(* Logix 5000 project; controller Drives_Line1 1756-L72 rev 20.13; software revision 20.04; part 5 of 21 *)
(* tags used below, declared in another part *)
   Diamtest : BOOL;
   Diamtest_mm : REAL;
   TimeForBr : TIMER;
   TimeOffFan : TIMER;
   TonRefOn : TIMER;
   Unwinder_1_DiamCalcOn : BOOL;
   Unwinder_1_JEC : REAL;
   Unwinder_1_JLossCrvSpd : REAL[21];
   Unwinder_1_JMaterial : REAL;
   Unwinder_1_LossCrvTrq_Pct : REAL[21];
   Unwinder_1_MatMass : REAL;
   Unwinder_1_MatVolume : REAL;
   Unwinder_1_MaxMass : REAL;
   Unwinder_1_MaxVolume : REAL;
   Unwinder_1_PctPerN : REAL;
   Unwinder_1_RatedTrq : REAL;
   Unwinder_1_RPMPerMPS : REAL;
   Unwinder_1_Running : BOOL;
   Unwinder_1_SpdMps_Flt : REAL;
   Unwinder_1_SpdRpm_Flt : REAL;
   zUnwinder_1_JGainQ1Q2 : REAL;
   zUnwinder_1_JGainQ3Q4 : REAL;
   zUnwinder_1_RateMax : REAL;
   zUnwinder_1_SpdReg_BWMax : REAL;
   zUnwinder_1_SpdReg_BWmin : REAL;
   zUnwinder_1_Stall_Spd : REAL;
   zUnwinder_1_TenRefRate : REAL;
   zUnwinder_1_TenSpStall : REAL;
   zUnwinder_1_TrqTrimLimMax_Pct : REAL;
   zUnwinder_1_TrqTrimLimMin_Pct : REAL;
   Bridle_01 : UDT_Bridle_3M;
   EntryConfig : UDT_Config_Zone;
   EntryCtrl : UDT_Control_Zone;
   LineSetpoints : UDT_Setpoints_Line;
   Unwinder_1 : UDT_Unwinder;
   Winder : UDT_Winder;
   zPi : REAL;
(* P10_Unwinder_1, continued *)

ROUTINE R05_Control   (* ladder *)
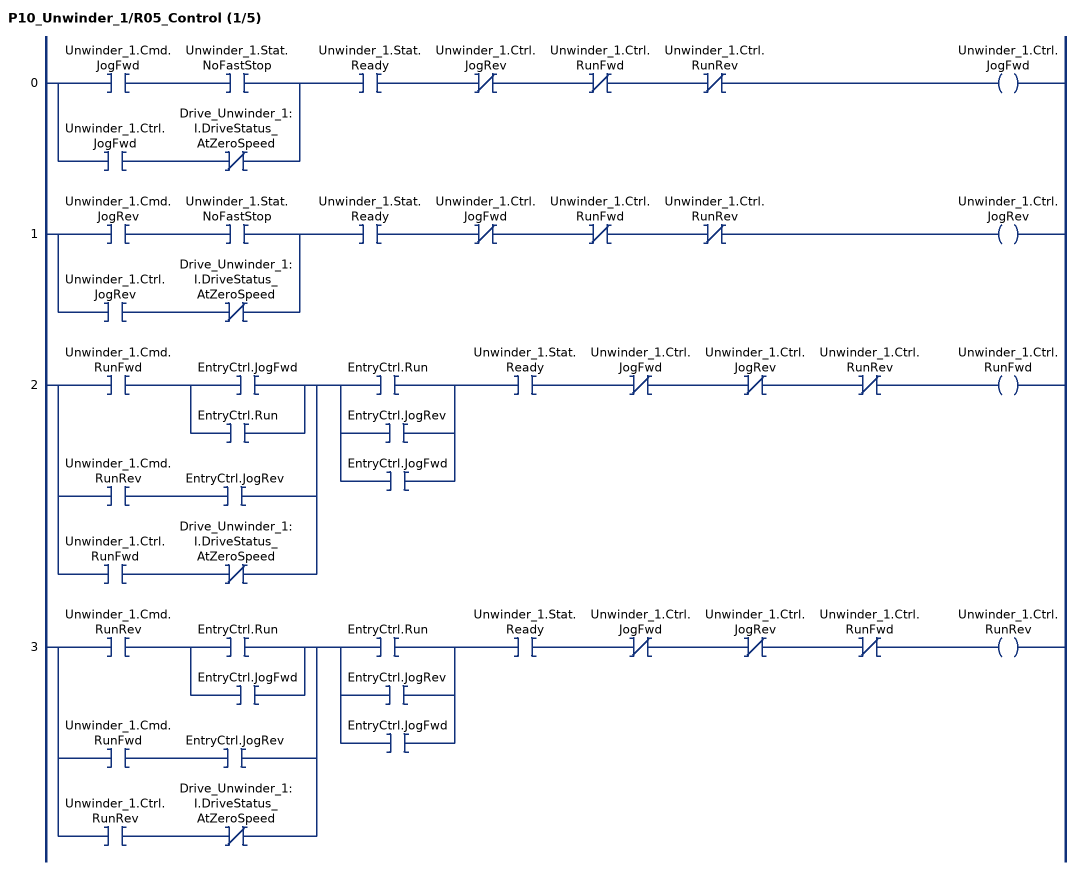
   0: [XIC(Unwinder_1.Cmd.JogFwd) XIC(Unwinder_1.Stat.NoFastStop) ,XIC(Unwinder_1.Ctrl.JogFwd) XIO(Drive_Unwinder_1:I.DriveStatus_AtZeroSpeed) ]XIC(Unwinder_1.Stat.Ready)XIO(Unwinder_1.Ctrl.JogRev)XIO(Unwinder_1.Ctrl.RunFwd)XIO(Unwinder_1.Ctrl.RunRev)OTE(Unwinder_1.Ctrl.JogFwd);
   1: [XIC(Unwinder_1.Cmd.JogRev) XIC(Unwinder_1.Stat.NoFastStop) ,XIC(Unwinder_1.Ctrl.JogRev) XIO(Drive_Unwinder_1:I.DriveStatus_AtZeroSpeed) ]XIC(Unwinder_1.Stat.Ready)XIO(Unwinder_1.Ctrl.JogFwd)XIO(Unwinder_1.Ctrl.RunFwd)XIO(Unwinder_1.Ctrl.RunRev)OTE(Unwinder_1.Ctrl.JogRev);
   2: [XIC(Unwinder_1.Cmd.RunFwd) [XIC(EntryCtrl.JogFwd) ,XIC(EntryCtrl.Run) ] ,XIC(Unwinder_1.Cmd.RunRev) XIC(EntryCtrl.JogRev) ,XIC(Unwinder_1.Ctrl.RunFwd) XIO(Drive_Unwinder_1:I.DriveStatus_AtZeroSpeed) ][XIC(EntryCtrl.Run) ,XIC(EntryCtrl.JogRev) ,XIC(EntryCtrl.JogFwd) ]XIC(Unwinder_1.Stat.Ready)XIO(Unwinder_1.Ctrl.JogFwd)XIO(Unwinder_1.Ctrl.JogRev)XIO(Unwinder_1.Ctrl.RunRev)OTE(Unwinder_1.Ctrl.RunFwd);
   3: [XIC(Unwinder_1.Cmd.RunRev) [XIC(EntryCtrl.Run) ,XIC(EntryCtrl.JogFwd) ] ,XIC(Unwinder_1.Cmd.RunFwd) XIC(EntryCtrl.JogRev) ,XIC(Unwinder_1.Ctrl.RunRev) XIO(Drive_Unwinder_1:I.DriveStatus_AtZeroSpeed) ][XIC(EntryCtrl.Run) ,XIC(EntryCtrl.JogRev) ,XIC(EntryCtrl.JogFwd) ]XIC(Unwinder_1.Stat.Ready)XIO(Unwinder_1.Ctrl.JogFwd)XIO(Unwinder_1.Ctrl.JogRev)XIO(Unwinder_1.Ctrl.RunFwd)OTE(Unwinder_1.Ctrl.RunRev);
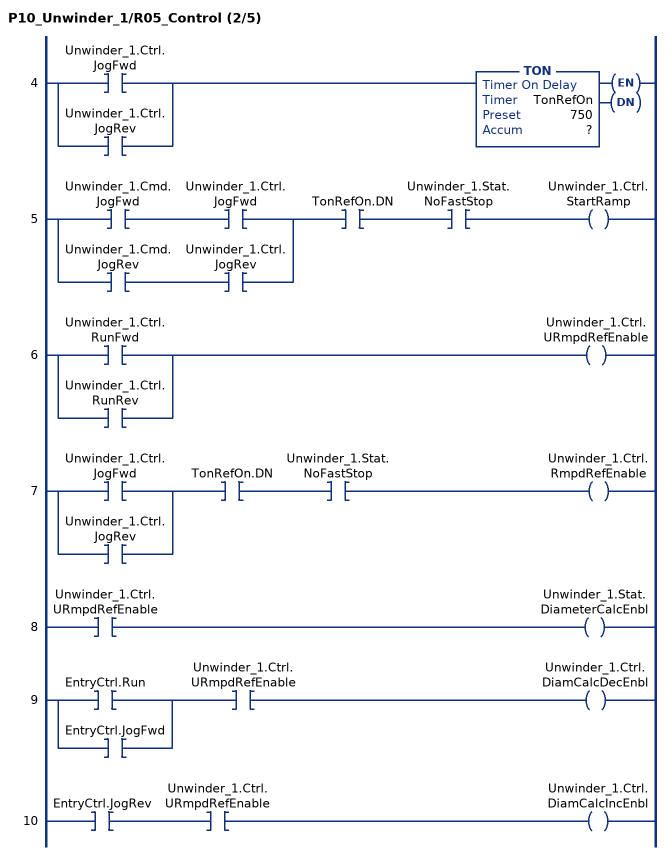
   4: [XIC(Unwinder_1.Ctrl.JogFwd) ,XIC(Unwinder_1.Ctrl.JogRev) ]TON(TonRefOn,?,?);
   5: [XIC(Unwinder_1.Cmd.JogFwd) XIC(Unwinder_1.Ctrl.JogFwd) ,XIC(Unwinder_1.Cmd.JogRev) XIC(Unwinder_1.Ctrl.JogRev) ]XIC(TonRefOn.DN)XIC(Unwinder_1.Stat.NoFastStop)OTE(Unwinder_1.Ctrl.StartRamp);
   6: [XIC(Unwinder_1.Ctrl.RunFwd) ,XIC(Unwinder_1.Ctrl.RunRev) ]OTE(Unwinder_1.Ctrl.URmpdRefEnable);
   7: [XIC(Unwinder_1.Ctrl.JogFwd) ,XIC(Unwinder_1.Ctrl.JogRev) ]XIC(TonRefOn.DN)XIC(Unwinder_1.Stat.NoFastStop)OTE(Unwinder_1.Ctrl.RmpdRefEnable);
   8: XIC(Unwinder_1.Ctrl.URmpdRefEnable)OTE(Unwinder_1.Stat.DiameterCalcEnbl);
   9: [XIC(EntryCtrl.Run) ,XIC(EntryCtrl.JogFwd) ]XIC(Unwinder_1.Ctrl.URmpdRefEnable)OTE(Unwinder_1.Ctrl.DiamCalcDecEnbl);
   10: XIC(EntryCtrl.JogRev)XIC(Unwinder_1.Ctrl.URmpdRefEnable)OTE(Unwinder_1.Ctrl.DiamCalcIncEnbl);
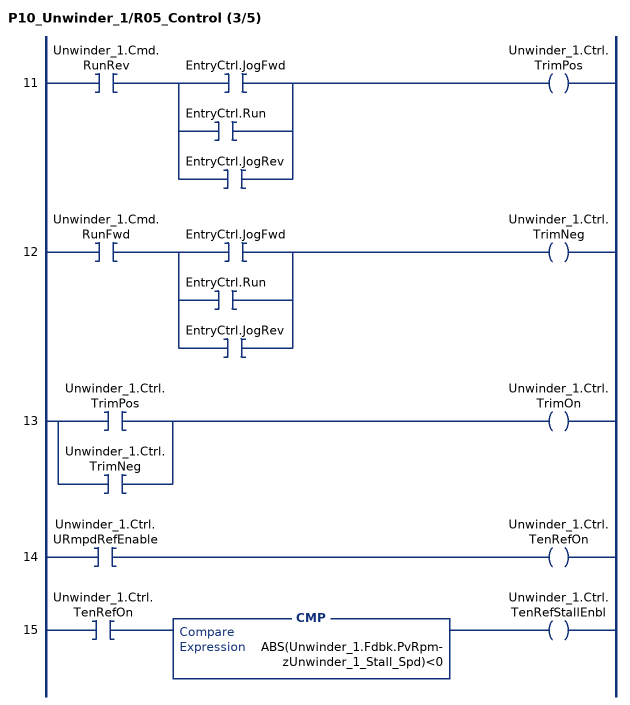
   11: XIC(Unwinder_1.Cmd.RunRev)[XIC(EntryCtrl.JogFwd) ,XIC(EntryCtrl.Run) ,XIC(EntryCtrl.JogRev) ]OTE(Unwinder_1.Ctrl.TrimPos);
   12: XIC(Unwinder_1.Cmd.RunFwd)[XIC(EntryCtrl.JogFwd) ,XIC(EntryCtrl.Run) ,XIC(EntryCtrl.JogRev) ]OTE(Unwinder_1.Ctrl.TrimNeg);
   13: [XIC(Unwinder_1.Ctrl.TrimPos) ,XIC(Unwinder_1.Ctrl.TrimNeg) ]OTE(Unwinder_1.Ctrl.TrimOn);
   14: XIC(Unwinder_1.Ctrl.URmpdRefEnable)OTE(Unwinder_1.Ctrl.TenRefOn);
   15: XIC(Unwinder_1.Ctrl.TenRefOn)CMP(ABS(Unwinder_1.Fdbk.PvRpm-zUnwinder_1_Stall_Spd)<0)OTE(Unwinder_1.Ctrl.TenRefStallEnbl);
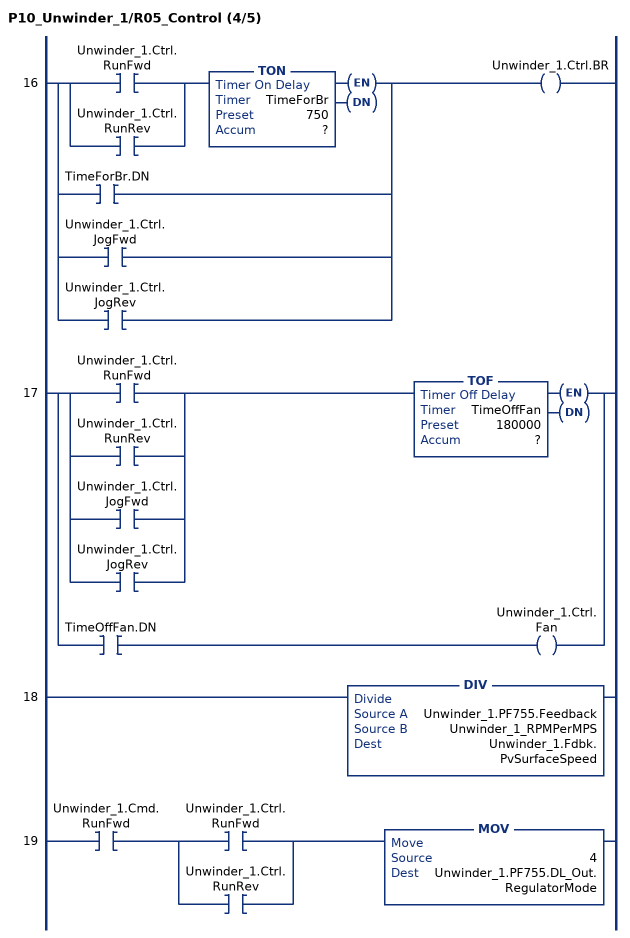
   16: [[XIC(Unwinder_1.Ctrl.RunFwd) ,XIC(Unwinder_1.Ctrl.RunRev) ] TON(TimeForBr,?,?) ,XIC(TimeForBr.DN) ,XIC(Unwinder_1.Ctrl.JogFwd) ,XIC(Unwinder_1.Ctrl.JogRev) ]OTE(Unwinder_1.Ctrl.BR);
   17: [[XIC(Unwinder_1.Ctrl.RunFwd) ,XIC(Unwinder_1.Ctrl.RunRev) ,XIC(Unwinder_1.Ctrl.JogFwd) ,XIC(Unwinder_1.Ctrl.JogRev) ] TOF(TimeOffFan,?,?) ,XIC(TimeOffFan.DN) OTE(Unwinder_1.Ctrl.Fan) ];
   18: DIV(Unwinder_1.PF755.Feedback,Unwinder_1_RPMPerMPS,Unwinder_1.Fdbk.PvSurfaceSpeed);
   19: XIC(Unwinder_1.Cmd.RunFwd)[XIC(Unwinder_1.Ctrl.RunFwd) ,XIC(Unwinder_1.Ctrl.RunRev) ]MOV(4,Unwinder_1.PF755.DL_Out.RegulatorMode);
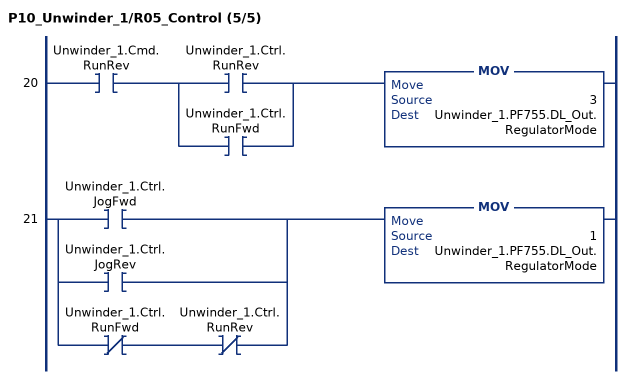
   20: XIC(Unwinder_1.Cmd.RunRev)[XIC(Unwinder_1.Ctrl.RunRev) ,XIC(Unwinder_1.Ctrl.RunFwd) ]MOV(3,Unwinder_1.PF755.DL_Out.RegulatorMode);
   21: [XIC(Unwinder_1.Ctrl.JogFwd) ,XIC(Unwinder_1.Ctrl.JogRev) ,XIO(Unwinder_1.Ctrl.RunFwd) XIO(Unwinder_1.Ctrl.RunRev) ]MOV(1,Unwinder_1.PF755.DL_Out.RegulatorMode);
END_ROUTINE

ROUTINE R07_TenFb   (* function block diagram *)
   SHEET 1   // Torque Feedback
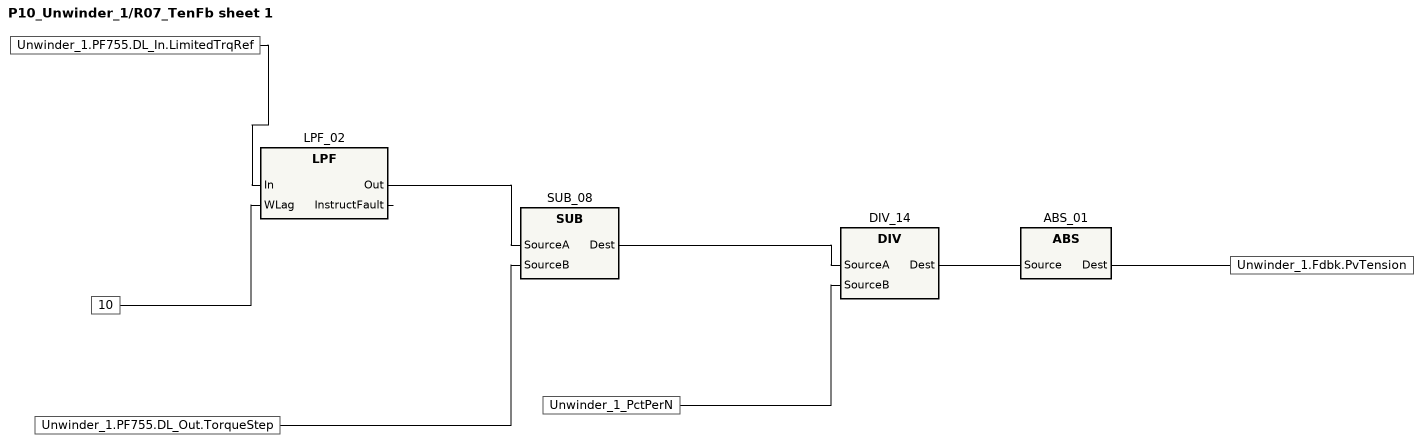
   LPF_02 : LPF(In := Unwinder_1.PF755.DL_In.LimitedTrqRef, WLag := 10);   // unwired pins: InstructFault
   SUB_08 : SUB(SourceA := LPF_02.Out, SourceB := Unwinder_1.PF755.DL_Out.TorqueStep);
   DIV_14 : DIV(SourceA := SUB_08.Dest, SourceB := Unwinder_1_PctPerN);
   ABS_01 : ABS(Source := DIV_14.Dest);
   Unwinder_1.Fdbk.PvTension := ABS_01.Dest;
   SHEET 2   // Speed Feedback
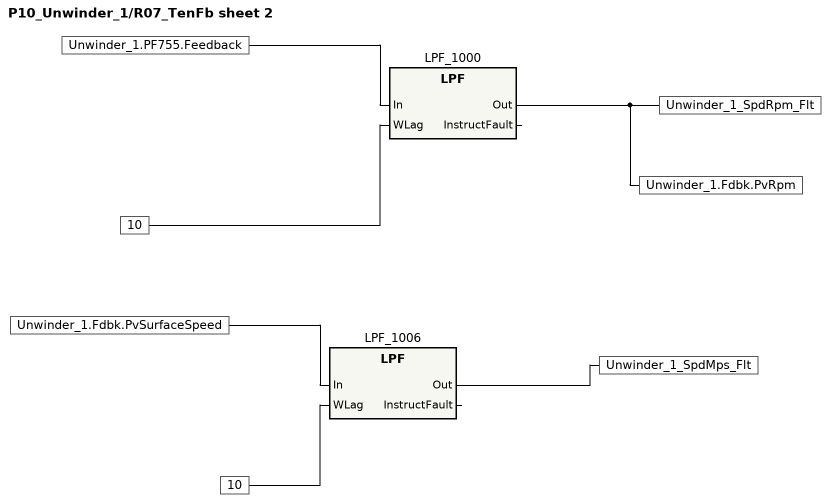
   LPF_1006 : LPF(In := Unwinder_1.Fdbk.PvSurfaceSpeed, WLag := 10);   // unwired pins: InstructFault
   LPF_1000 : LPF(In := Unwinder_1.PF755.Feedback, WLag := 10);   // unwired pins: InstructFault
   Unwinder_1_SpdMps_Flt := LPF_1006.Out;
   Unwinder_1.Fdbk.PvRpm := LPF_1000.Out;
   Unwinder_1_SpdRpm_Flt := LPF_1000.Out;
END_ROUTINE

ROUTINE R09_DiamCalc   (* function block diagram *)
   SHEET 1   // Distance/Angle Integration
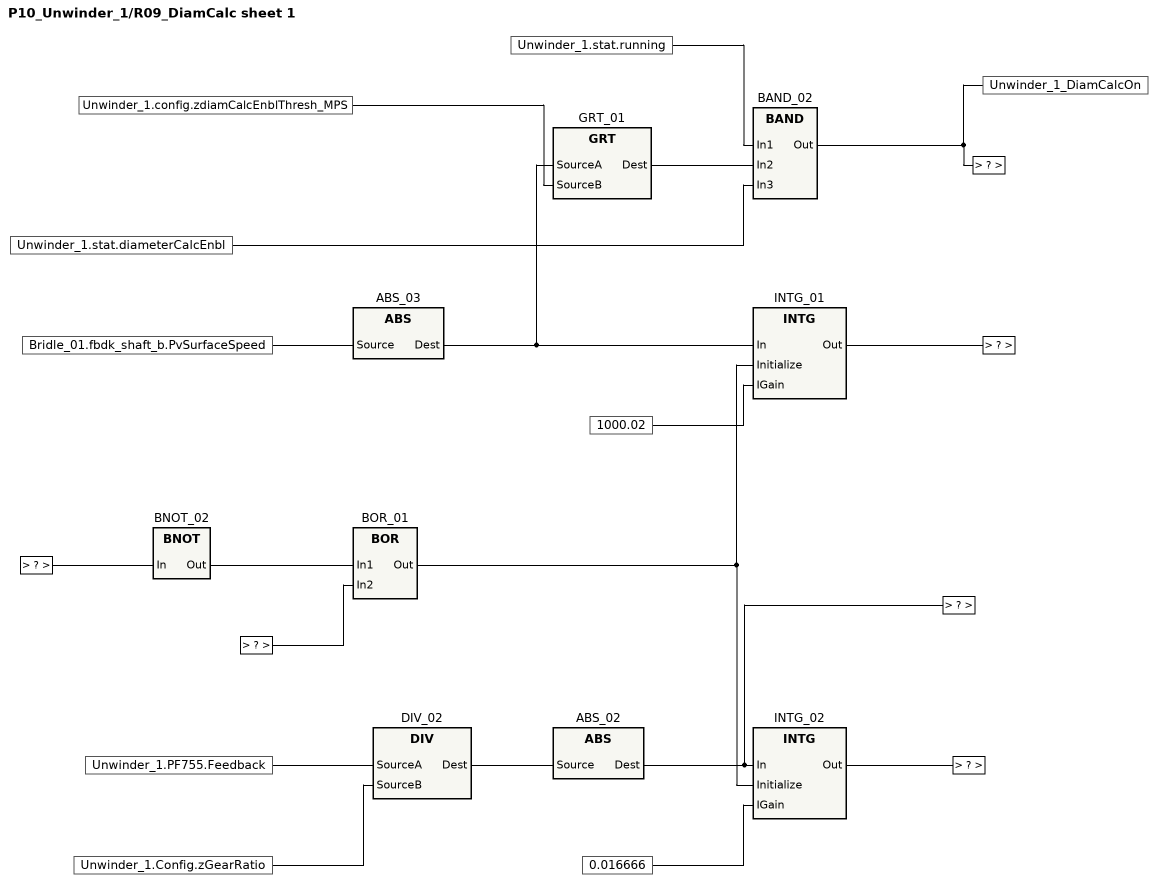
   ABS_03 : ABS(Source := Bridle_01.fbdk_shaft_b.PvSurfaceSpeed);
   DIV_02 : DIV(SourceA := Unwinder_1.PF755.Feedback, SourceB := Unwinder_1.Config.zGearRatio);
   GRT_01 : GRT(SourceA := ABS_03.Dest, SourceB := Unwinder_1.config.zdiamCalcEnblThresh_MPS);
   ABS_02 : ABS(Source := DIV_02.Dest);
   BAND_02 : BAND(In1 := Unwinder_1.stat.running, In2 := GRT_01.Dest, In3 := Unwinder_1.stat.diameterCalcEnbl);
   WIRE(?) := ABS_02.Dest;
   BNOT_02 : BNOT(In := WIRE(?));
   BOR_01 : BOR(In1 := BNOT_02.Out, In2 := WIRE(?) {feedback});
   INTG_01 : INTG(In := ABS_03.Dest, Initialize := BOR_01.Out, IGain := 1000.02);
   INTG_02 : INTG(In := ABS_02.Dest, Initialize := BOR_01.Out, IGain := 0.016666);
   WIRE(?) := INTG_02.Out;
   WIRE(?) := BAND_02.Out;
   Unwinder_1_DiamCalcOn := BAND_02.Out;
   WIRE(?) := INTG_01.Out;
   SHEET 2   // Diameter Calculate
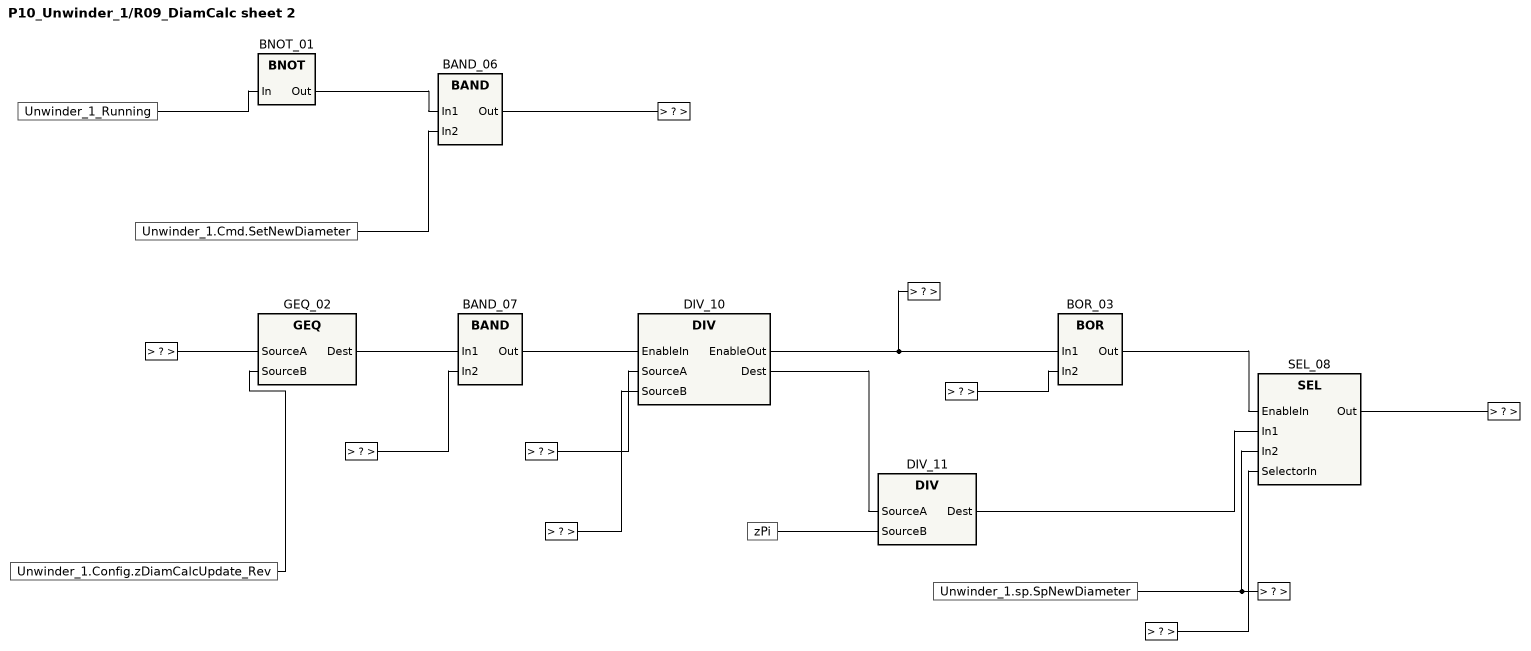
   BNOT_01 : BNOT(In := Unwinder_1_Running);
   BAND_06 : BAND(In1 := BNOT_01.Out, In2 := Unwinder_1.Cmd.SetNewDiameter);
   WIRE(?) := BAND_06.Out;
   WIRE(?) := Unwinder_1.sp.SpNewDiameter;
   GEQ_02 : GEQ(SourceA := WIRE(?), SourceB := Unwinder_1.Config.zDiamCalcUpdate_Rev);
   BAND_07 : BAND(In1 := GEQ_02.Dest, In2 := WIRE(?));
   DIV_10 : DIV(EnableIn := BAND_07.Out, SourceA := WIRE(?), SourceB := WIRE(?));
   DIV_11 : DIV(SourceA := DIV_10.Dest, SourceB := zPi);
   WIRE(?) := DIV_10.EnableOut;
   BOR_03 : BOR(In1 := DIV_10.EnableOut, In2 := WIRE(?));
   SEL_08 : SEL(EnableIn := BOR_03.Out, In1 := DIV_11.Dest, In2 := Unwinder_1.sp.SpNewDiameter, SelectorIn := WIRE(?));
   WIRE(?) := SEL_08.Out;
   SHEET 3   // Rate/Magnitude Limit
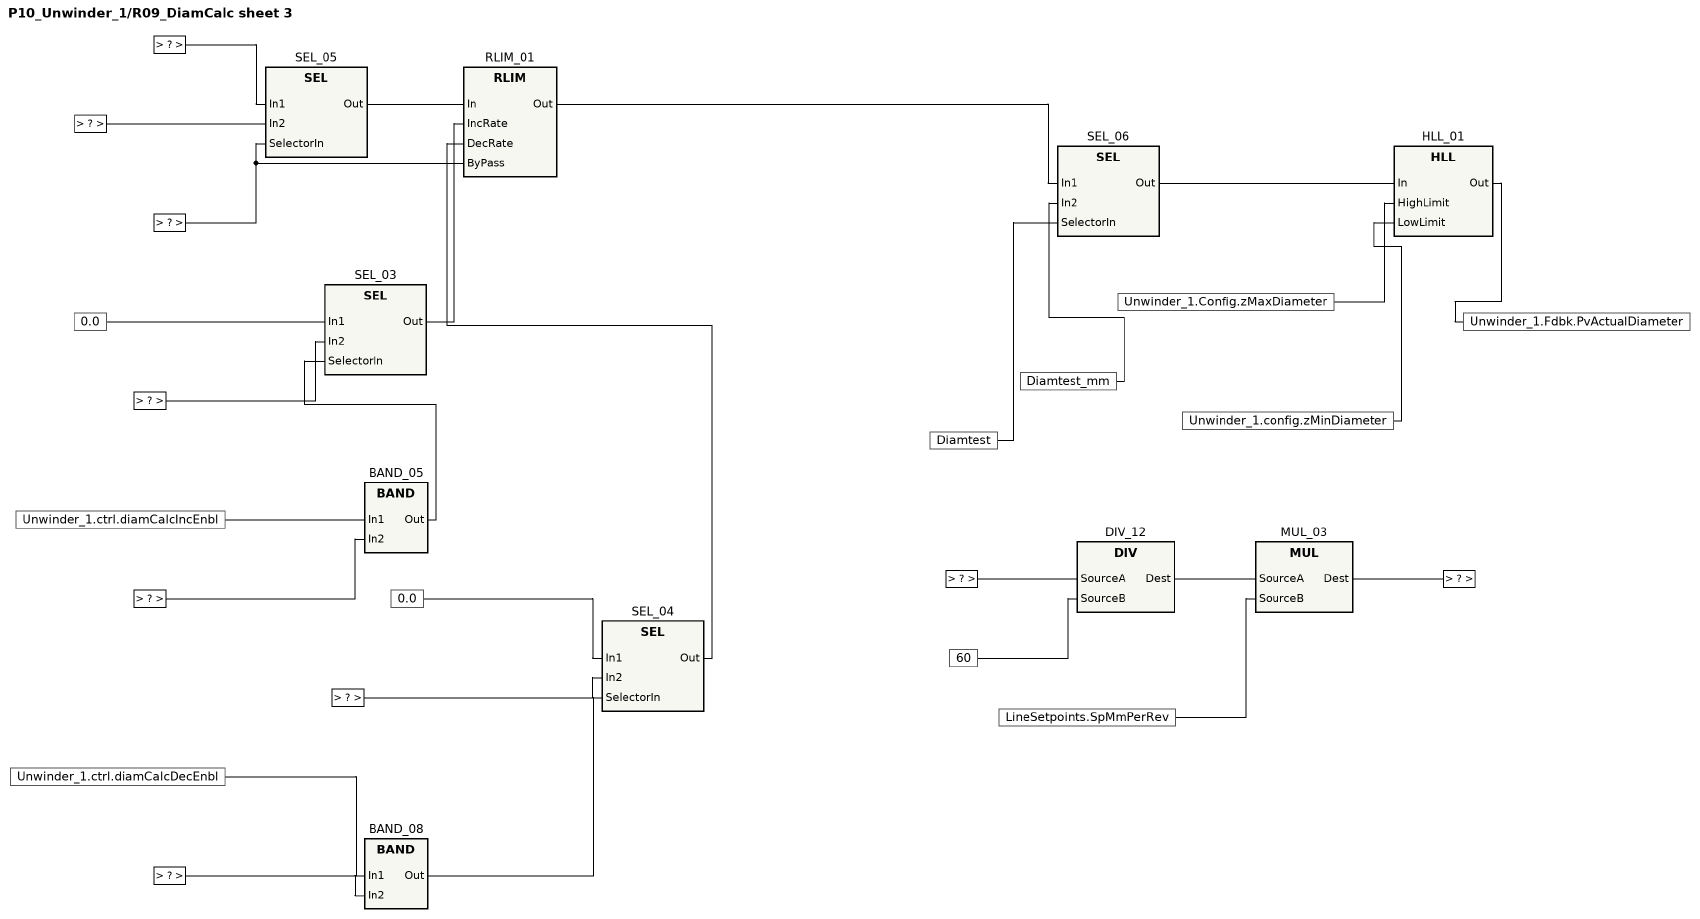
   BAND_05 : BAND(In1 := Unwinder_1.ctrl.diamCalcIncEnbl, In2 := WIRE(?));
   SEL_03 : SEL(In1 := 0.0, In2 := WIRE(?), SelectorIn := BAND_05.Out);
   SEL_05 : SEL(In1 := WIRE(?), In2 := WIRE(?), SelectorIn := WIRE(?));
   BAND_08 : BAND(In1 := Unwinder_1.ctrl.diamCalcDecEnbl, In2 := WIRE(?));
   SEL_04 : SEL(In1 := 0.0, In2 := WIRE(?), SelectorIn := BAND_08.Out);
   RLIM_01 : RLIM(In := SEL_05.Out, IncRate := SEL_03.Out, DecRate := SEL_04.Out, ByPass := WIRE(?));
   SEL_06 : SEL(In1 := RLIM_01.Out, In2 := Diamtest_mm, SelectorIn := Diamtest);
   HLL_01 : HLL(In := SEL_06.Out, HighLimit := Unwinder_1.Config.zMaxDiameter, LowLimit := Unwinder_1.config.zMinDiameter);
   Unwinder_1.Fdbk.PvActualDiameter := HLL_01.Out;
   DIV_12 : DIV(SourceA := WIRE(?), SourceB := 60);
   MUL_03 : MUL(SourceA := DIV_12.Dest, SourceB := LineSetpoints.SpMmPerRev);
   WIRE(?) := MUL_03.Dest;
END_ROUTINE

ROUTINE R10_Calculate   (* structured text *)
   // Calculate
   // Speed Conversion
   //
   // * * * * * * * * * * * * * * * * * * * * * * * * * * *
   //
   // Calculates conversion factor from surface speed [MPS] to rotational speeds [RPM].
   //
   //             Gear Ratio * 1000 [mm/M]
   // RPM/MPS =  -------------------------- * 60
   //             Roll Diameter [mm] * PI
   //
   Unwinder_1_RPMPerMPS := (Unwinder_1.Config.zGearRatio * 1000.0) / (Unwinder_1.Fdbk.PvActualDiameter * zPi) * 60;
   //
   // * * * * * * * * * * * * * * * * * * * * * * * * * * *
   //
   // Calculate
   // (Rated Motor Torque)
   //
   // * * * * * * * * * * * * * * * * * * * * * * * * * * *
   //
   //                       MtrPwrRated [KW] * 9549
   // MtrTrqRated_Nm = ----------------------------
   //                           MtrSpdBase [RPM]
   //
   Unwinder_1_RatedTrq := Unwinder_1.Config.zMotorPwr * 9549 / Unwinder_1.Config.zMtrBaseSpd;
   //
   
   
   //
   // Calculate
   // (Center Winder Inertia)
   //
   // * * * * * * * * * * * * * * * * * * * * * * * * * * *
   //
   // MaterialVolume_m3 = (Pi * (Diam_mm/2000)**2 - Pi * (DiamMinEC_mm/2000)**2) * Width_mm/1000
   //
   Unwinder_1_MatVolume := (zPi * (Unwinder_1.Fdbk.PvActualDiameter/2000)**2)
   - (zPi * (Unwinder_1.Config.zMinDiameter/2000)**2)* (LineSetpoints.WebWidth  / 1000);
   Unwinder_1_MaxVolume:= (zPi * (Unwinder_1.Config.zMaxDiameter/2000)**2)* LineSetpoints.WebWidth / 1000;
   // MaterialMass_Kg = MaterialVolume_m3 * Density_Kgm3
   //
   Unwinder_1_MatMass := Unwinder_1_MatVolume * LineSetpoints.MaterialDensity ;
   Unwinder_1_MaxMass:= Unwinder_1_MaxVolume * LineSetpoints.MaterialDensity ;
   //
   // JMaterial_Kgm2 = MaterialWeight_Kg / 2 * ((Diam_mm/2000)**2 + (DiamMinEC_mm/2000)**2) / GearRatio**2
   //
   Unwinder_1_JMaterial := Unwinder_1_MatMass / 2 *
   ((Unwinder_1.Fdbk.PvActualDiameter/2000)**2 + (Unwinder_1.Config.zMinDiameter/2000)**2)
    / Unwinder_1.Config.zGearRatio**2 ;
   //
   // Calculate total reflected inertia [kilogram-meters**2]
   //
   Unwinder_1.Fdbk.PvTotalInertia := Unwinder_1_JEC + Unwinder_1_JMaterial ;
   //
   // * * * * * * * * * * * * * * * * * * * * * * * * * * *
   //
   // Calculate
   // (Normalized Inertia)
   //
   // * * * * * * * * * * * * * * * * * * * * * * * * * * *
   //
   //         J [Kgm**2] * MtrSpdBase [RPM]
   // J_Sec = -------------------------------
   //           9.549 * MtrTrqRated [Nm]
   //
   Unwinder_1.Fdbk.PvNormInertia := (Unwinder_1.Fdbk.PvTotalInertia * Unwinder_1.Config.zMtrBaseSpd)
   / (9.549 * Unwinder_1_RatedTrq);
   
   (*                         Diam [mm]           100                  1      *)
   (* Conversion_PctPerN =  ----------- * -------------------- * ----------- *)
   (*                         1000 * 2       MtrTrqRated [Nm]      GearRatio  *)
   
   Unwinder_1_PctPerN := Unwinder_1.Fdbk.PvActualDiameter / Unwinder_1.Config.zGearRatio
    / Unwinder_1_RatedTrq / 20.0 ;
END_ROUTINE

ROUTINE R11_TenRef   (* function block diagram *)
   SHEET 1   // Tension Reference
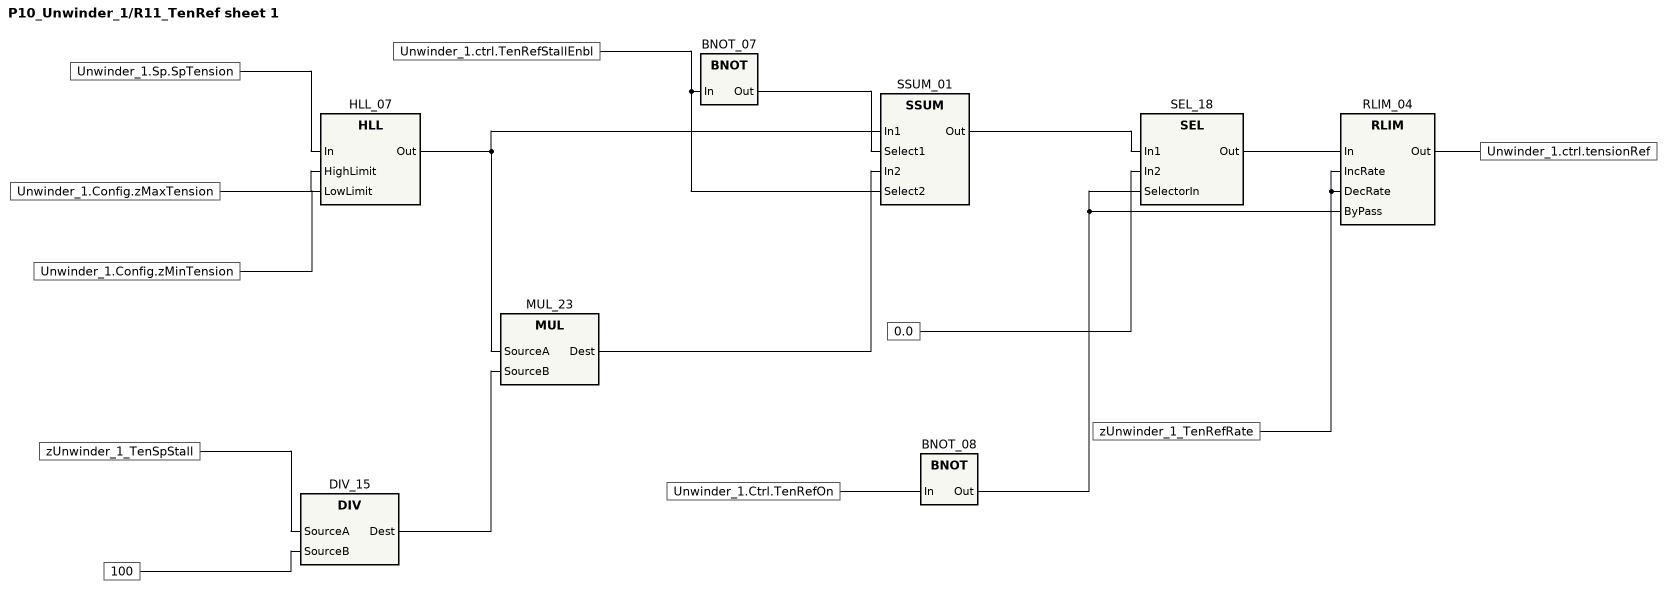
   DIV_15 : DIV(SourceA := zUnwinder_1_TenSpStall, SourceB := 100);
   HLL_07 : HLL(In := Unwinder_1.Sp.SpTension, HighLimit := Unwinder_1.Config.zMaxTension, LowLimit := Unwinder_1.Config.zMinTension);
   MUL_23 : MUL(SourceA := HLL_07.Out, SourceB := DIV_15.Dest);
   BNOT_07 : BNOT(In := Unwinder_1.ctrl.TenRefStallEnbl);
   SSUM_01 : SSUM(In1 := HLL_07.Out, Select1 := BNOT_07.Out, In2 := MUL_23.Dest, Select2 := Unwinder_1.ctrl.TenRefStallEnbl);
   BNOT_08 : BNOT(In := Unwinder_1.Ctrl.TenRefOn);
   SEL_18 : SEL(In1 := SSUM_01.Out, In2 := 0.0, SelectorIn := BNOT_08.Out);
   RLIM_04 : RLIM(In := SEL_18.Out, IncRate := zUnwinder_1_TenRefRate, DecRate := zUnwinder_1_TenRefRate, ByPass := BNOT_08.Out);
   Unwinder_1.ctrl.tensionRef := RLIM_04.Out;
END_ROUTINE

ROUTINE R12_DriveRef   (* function block diagram *)
   SHEET 1   // Jog reference
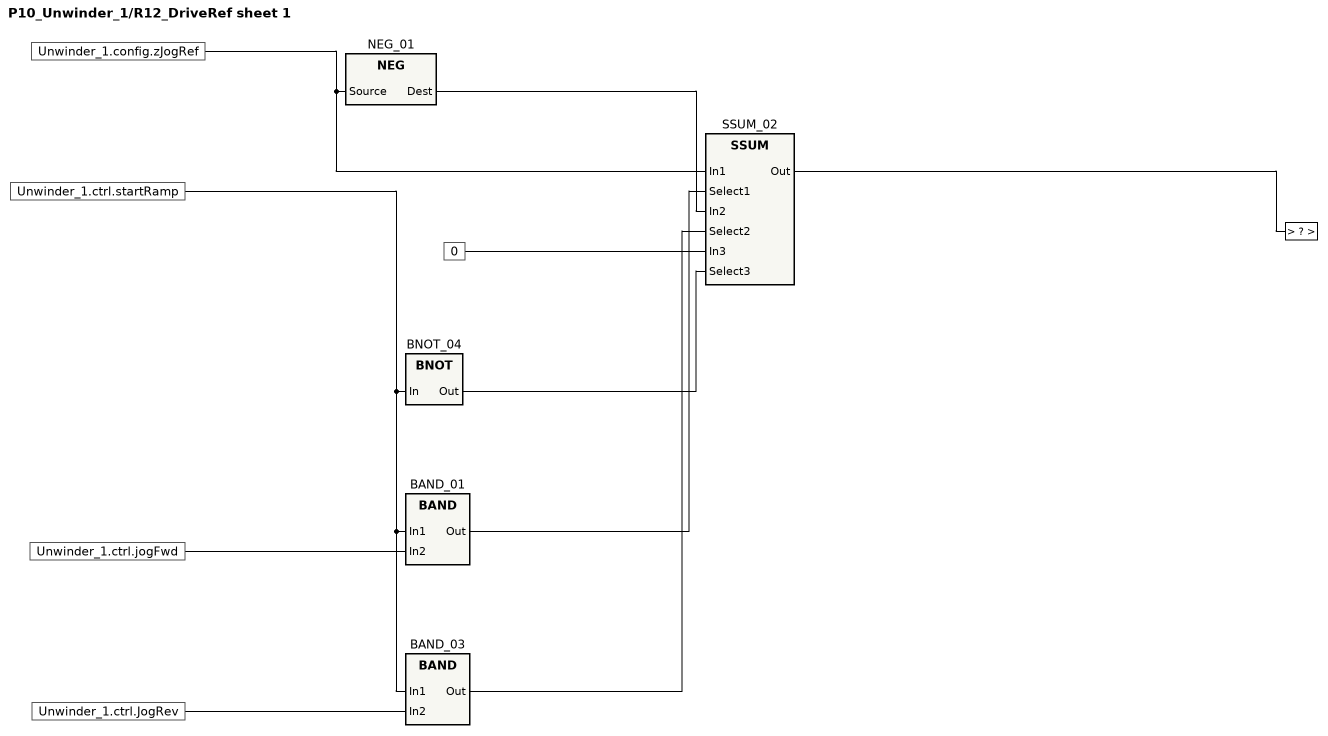
   NEG_01 : NEG(Source := Unwinder_1.config.zJogRef);
   BNOT_04 : BNOT(In := Unwinder_1.ctrl.startRamp);
   BAND_01 : BAND(In1 := Unwinder_1.ctrl.startRamp, In2 := Unwinder_1.ctrl.jogFwd);
   BAND_03 : BAND(In1 := Unwinder_1.ctrl.startRamp, In2 := Unwinder_1.ctrl.JogRev);
   SSUM_02 : SSUM(In1 := Unwinder_1.config.zJogRef, Select1 := BAND_01.Out, In2 := NEG_01.Dest, Select2 := BAND_03.Out, In3 := 0, Select3 := BNOT_04.Out);
   WIRE(?) := SSUM_02.Out;
   SHEET 2   // S-Curve
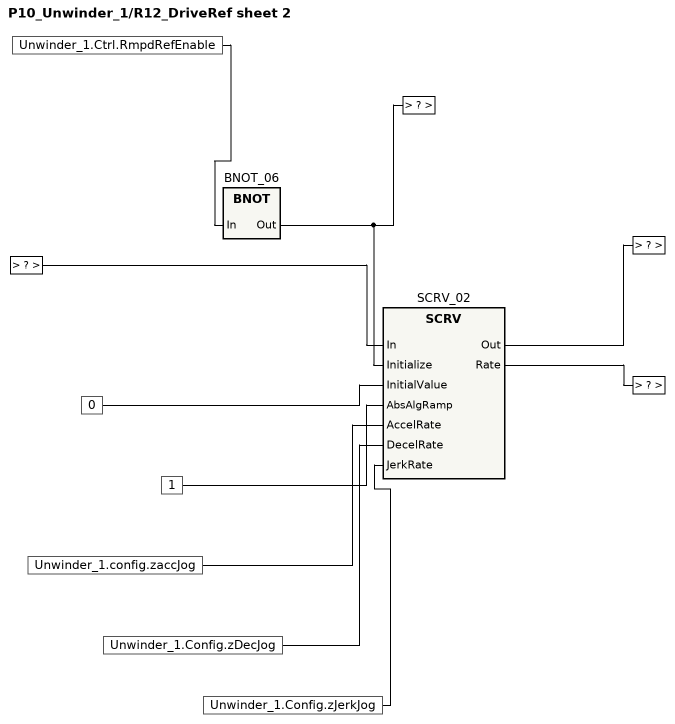
   BNOT_06 : BNOT(In := Unwinder_1.Ctrl.RmpdRefEnable);
   WIRE(?) := BNOT_06.Out;
   SCRV_02 : SCRV(In := WIRE(?), Initialize := BNOT_06.Out, InitialValue := 0, AbsAlgRamp := 1, AccelRate := Unwinder_1.config.zaccJog, DecelRate := Unwinder_1.Config.zDecJog, JerkRate := Unwinder_1.Config.zJerkJog);
   WIRE(?) := SCRV_02.Out;
   WIRE(?) := SCRV_02.Rate;
   SHEET 3   // Select ramped/unramped reference
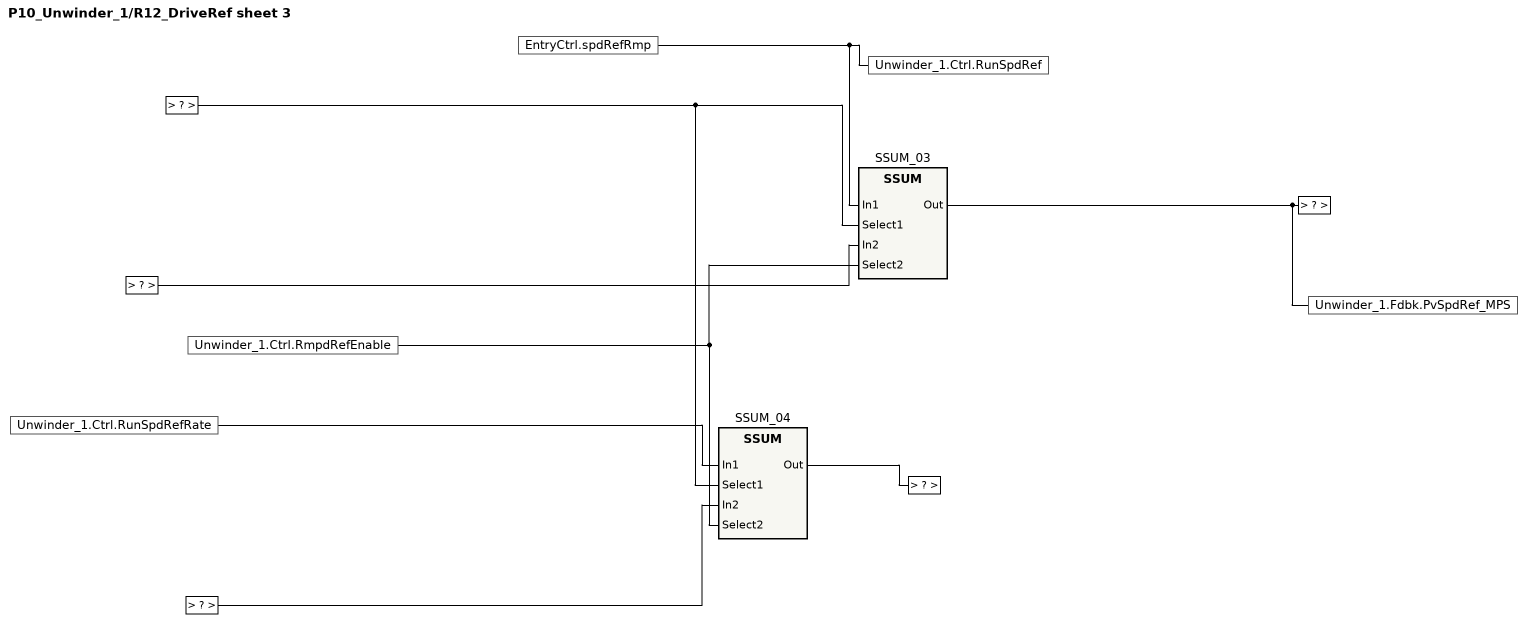
   Unwinder_1.Ctrl.RunSpdRef := EntryCtrl.spdRefRmp;
   SSUM_03 : SSUM(In1 := EntryCtrl.spdRefRmp, Select1 := WIRE(?), In2 := WIRE(?), Select2 := Unwinder_1.Ctrl.RmpdRefEnable);
   WIRE(?) := SSUM_03.Out;
   SSUM_04 : SSUM(In1 := Unwinder_1.Ctrl.RunSpdRefRate, Select1 := WIRE(?), In2 := WIRE(?), Select2 := Unwinder_1.Ctrl.RmpdRefEnable);
   WIRE(?) := SSUM_04.Out;
   Unwinder_1.Fdbk.PvSpdRef_MPS := SSUM_03.Out;
   SHEET 4   // Inertia Compensation
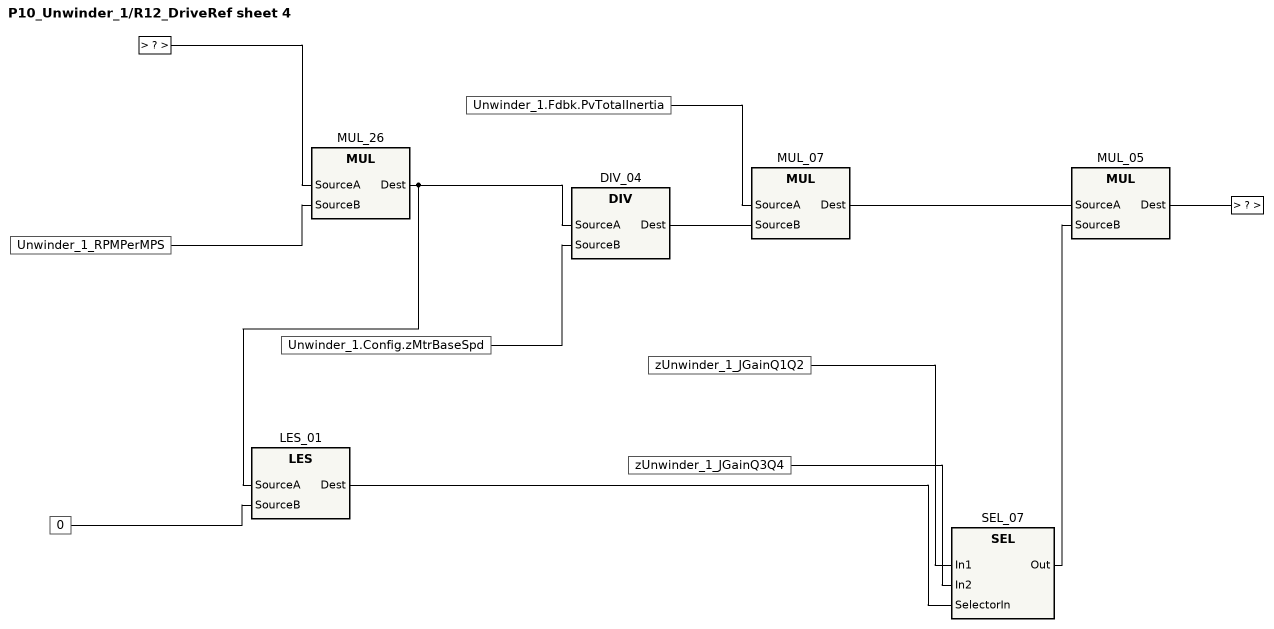
   MUL_26 : MUL(SourceA := WIRE(?), SourceB := Unwinder_1_RPMPerMPS);
   LES_01 : LES(SourceA := MUL_26.Dest, SourceB := 0);
   DIV_04 : DIV(SourceA := MUL_26.Dest, SourceB := Unwinder_1.Config.zMtrBaseSpd);
   MUL_07 : MUL(SourceA := Unwinder_1.Fdbk.PvTotalInertia, SourceB := DIV_04.Dest);
   SEL_07 : SEL(In1 := zUnwinder_1_JGainQ1Q2, In2 := zUnwinder_1_JGainQ3Q4, SelectorIn := LES_01.Dest);
   MUL_05 : MUL(SourceA := MUL_07.Dest, SourceB := SEL_07.Out);
   WIRE(?) := MUL_05.Dest;
   SHEET 5   // Friction and Windage Compensation
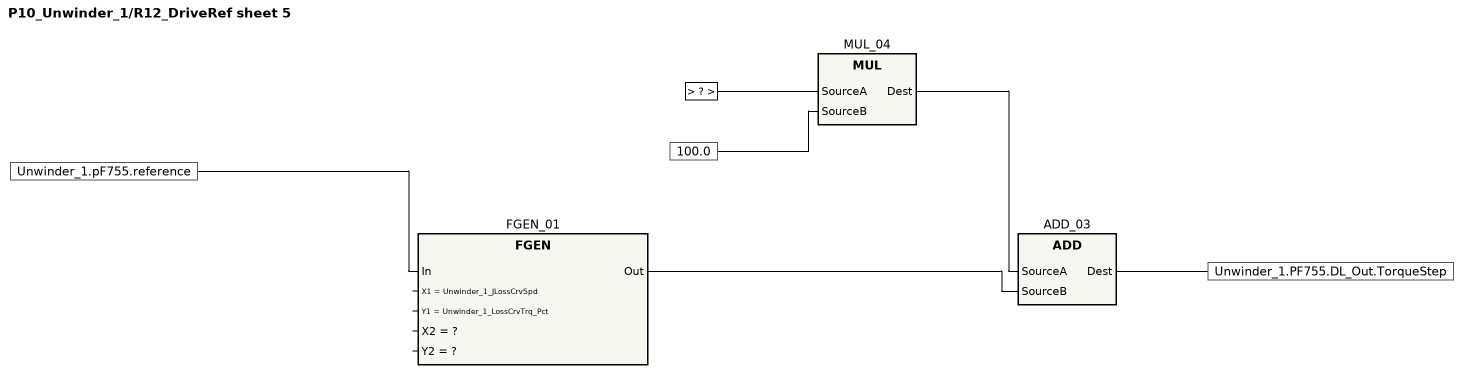
   FGEN_01 : FGEN(In := Unwinder_1.pF755.reference, X1 := Unwinder_1_JLossCrvSpd, Y1 := Unwinder_1_LossCrvTrq_Pct, X2 := ?, Y2 := ?);
   MUL_04 : MUL(SourceA := WIRE(?), SourceB := 100.0);
   ADD_03 : ADD(SourceA := MUL_04.Dest, SourceB := FGEN_01.Out);
   Unwinder_1.PF755.DL_Out.TorqueStep := ADD_03.Dest;
   SHEET 6   // Speed trim
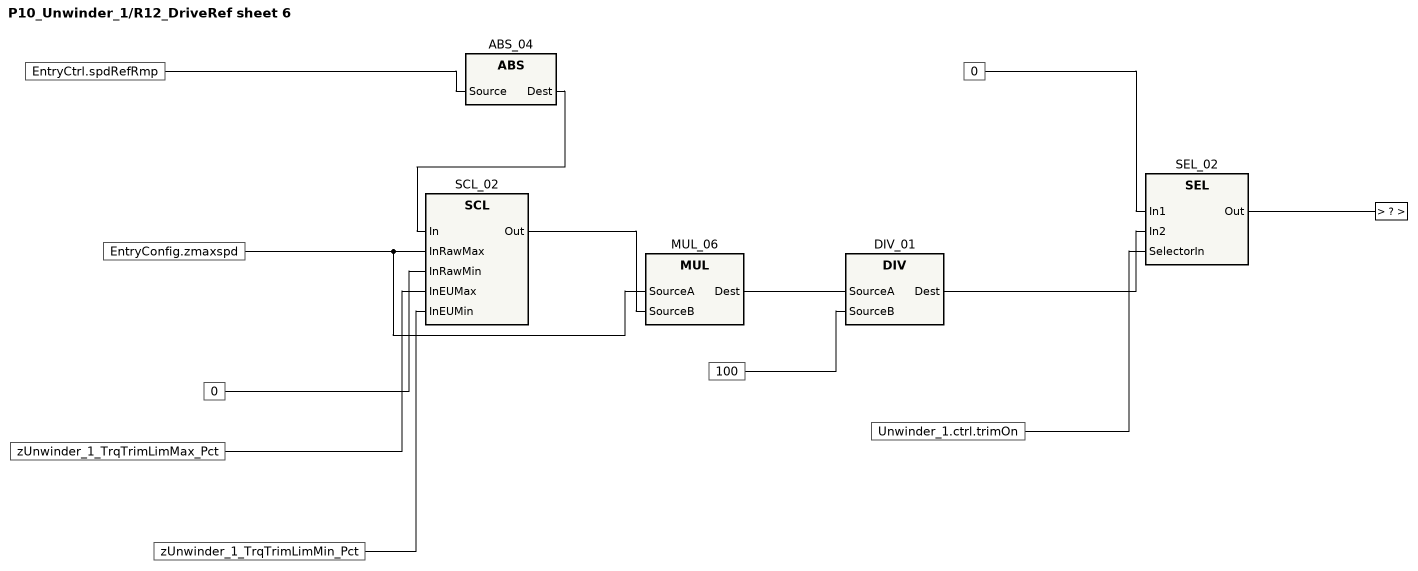
   ABS_04 : ABS(Source := EntryCtrl.spdRefRmp);
   SCL_02 : SCL(In := ABS_04.Dest, InRawMax := EntryConfig.zmaxspd, InRawMin := 0, InEUMax := zUnwinder_1_TrqTrimLimMax_Pct, InEUMin := zUnwinder_1_TrqTrimLimMin_Pct);
   MUL_06 : MUL(SourceA := EntryConfig.zmaxspd, SourceB := SCL_02.Out);
   DIV_01 : DIV(SourceA := MUL_06.Dest, SourceB := 100);
   SEL_02 : SEL(In1 := 0, In2 := DIV_01.Dest, SelectorIn := Unwinder_1.ctrl.trimOn);
   WIRE(?) := SEL_02.Out;
   SHEET 7   // Final speed reference
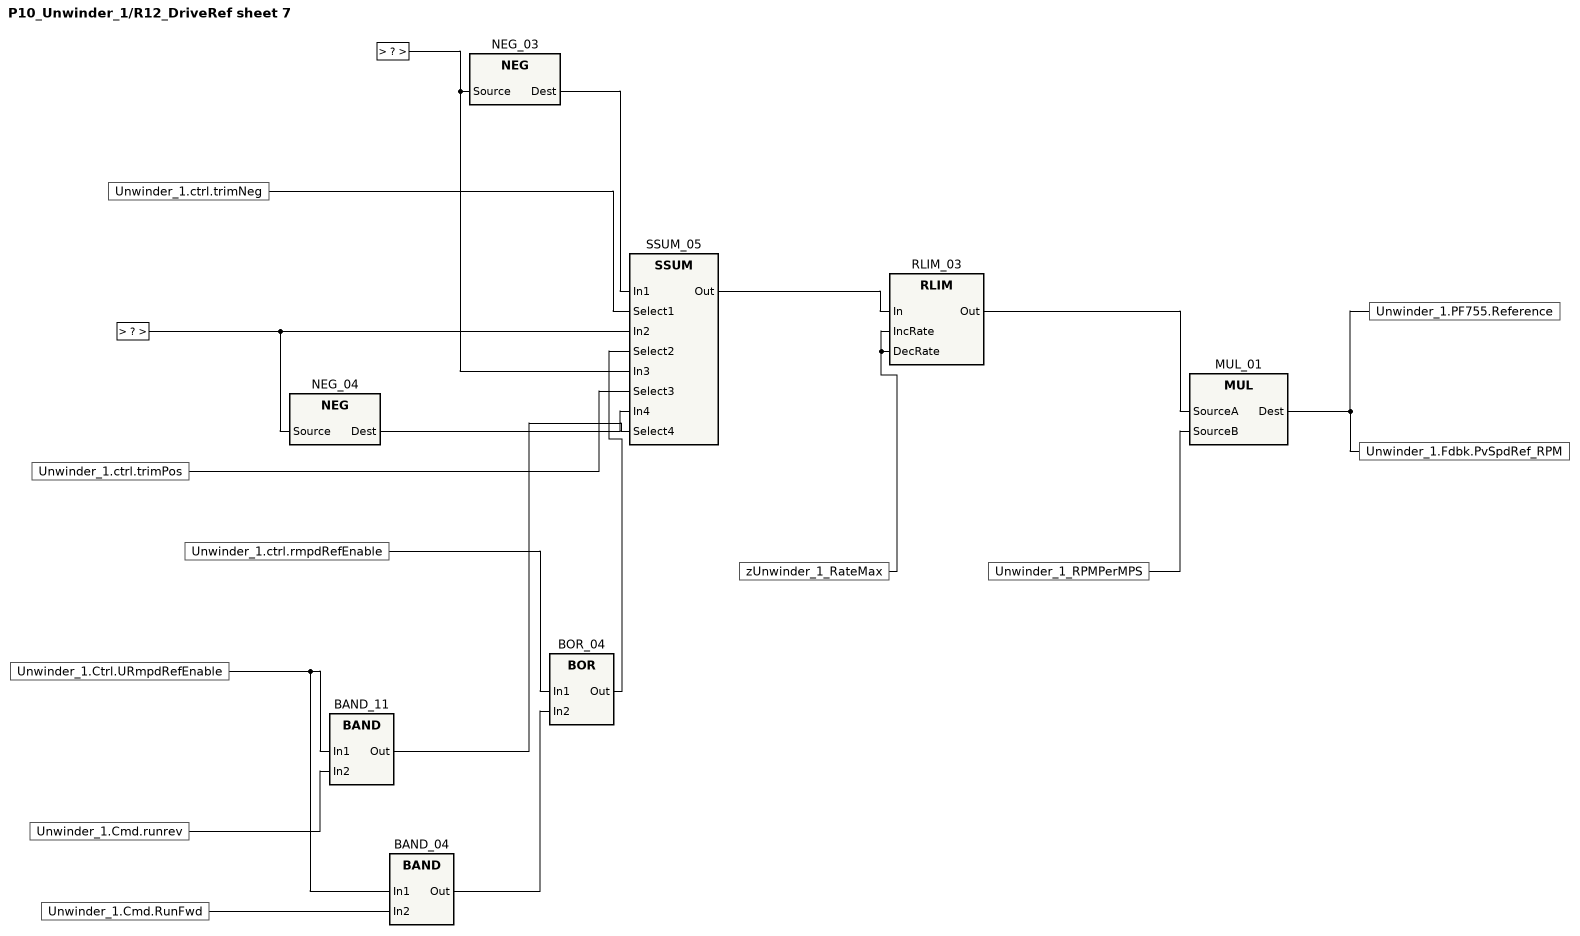
   NEG_04 : NEG(Source := WIRE(?));
   BAND_11 : BAND(In1 := Unwinder_1.Ctrl.URmpdRefEnable, In2 := Unwinder_1.Cmd.runrev);
   BAND_04 : BAND(In1 := Unwinder_1.Ctrl.URmpdRefEnable, In2 := Unwinder_1.Cmd.RunFwd);
   NEG_03 : NEG(Source := WIRE(?));
   BOR_04 : BOR(In1 := Unwinder_1.ctrl.rmpdRefEnable, In2 := BAND_04.Out);
   SSUM_05 : SSUM(In1 := NEG_03.Dest, Select1 := Unwinder_1.ctrl.trimNeg, In2 := WIRE(?), Select2 := BOR_04.Out, In3 := WIRE(?), Select3 := Unwinder_1.ctrl.trimPos, In4 := NEG_04.Dest, Select4 := BAND_11.Out);
   RLIM_03 : RLIM(In := SSUM_05.Out, IncRate := zUnwinder_1_RateMax, DecRate := zUnwinder_1_RateMax);
   MUL_01 : MUL(SourceA := RLIM_03.Out, SourceB := Unwinder_1_RPMPerMPS);
   Unwinder_1.Fdbk.PvSpdRef_RPM := MUL_01.Dest;
   Unwinder_1.PF755.Reference := MUL_01.Dest;
   SHEET 8   // Torque reference
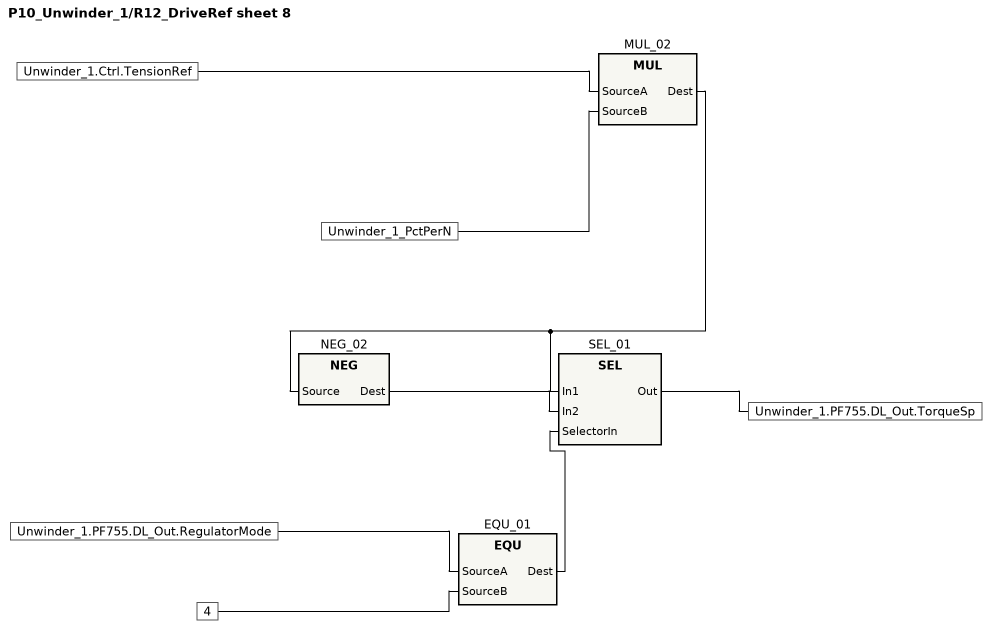
   EQU_01 : EQU(SourceA := Unwinder_1.PF755.DL_Out.RegulatorMode, SourceB := 4);
   MUL_02 : MUL(SourceA := Unwinder_1.Ctrl.TensionRef, SourceB := Unwinder_1_PctPerN);
   NEG_02 : NEG(Source := MUL_02.Dest);
   SEL_01 : SEL(In1 := MUL_02.Dest, In2 := NEG_02.Dest, SelectorIn := EQU_01.Dest);
   Unwinder_1.PF755.DL_Out.TorqueSp := SEL_01.Out;
   SHEET 9   // Speed regulator bandwidt
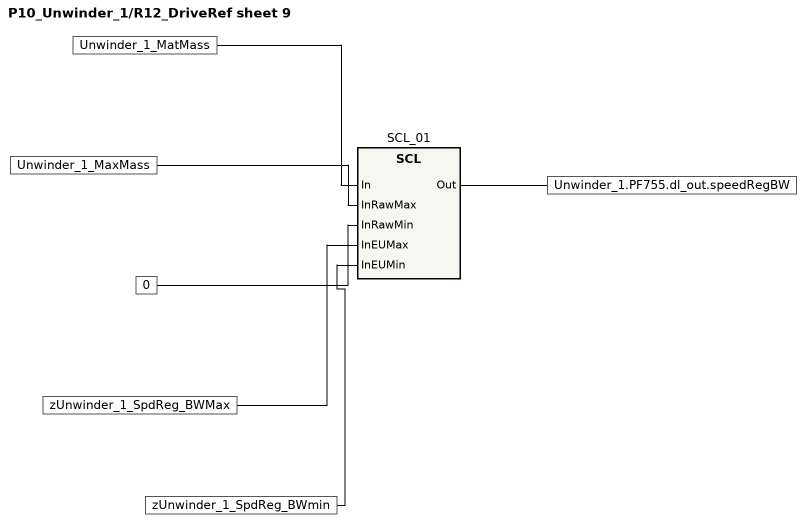
   SCL_01 : SCL(In := Unwinder_1_MatMass, InRawMax := Unwinder_1_MaxMass, InRawMin := 0, InEUMax := zUnwinder_1_SpdReg_BWMax, InEUMin := zUnwinder_1_SpdReg_BWmin);
   Unwinder_1.PF755.dl_out.speedRegBW := SCL_01.Out;
END_ROUTINE
